SYSTEM Test_7 (* System Configuration *)
  (* Standard: 61499-1 *)
  (* Version 0.3, 2003-12-05, JHC, Rockwell Automation, Renamed from NEWSYSTEM. *)
  (* Version 0.2, 2002-11-05, JHC, Rockwell Automation, Fixed missing (empty) FBD in Application. *)
  (* Version 0.1, 2002-01-17, JHC, Rockwell Automation, Minor cleanup *)
  (* Version 0.0, 2000-05-27, JHC, Rockwell Automation *)
  APPLICATION APP1
  END_APPLICATION
  DEVICE DEV1 : FRAME_DEVICE(BOUNDS := [300,300,300,300], GRID := [1,1])
    RESOURCE RES1 : PANEL_RESOURCE(ROWS := 1, COLS := 1)
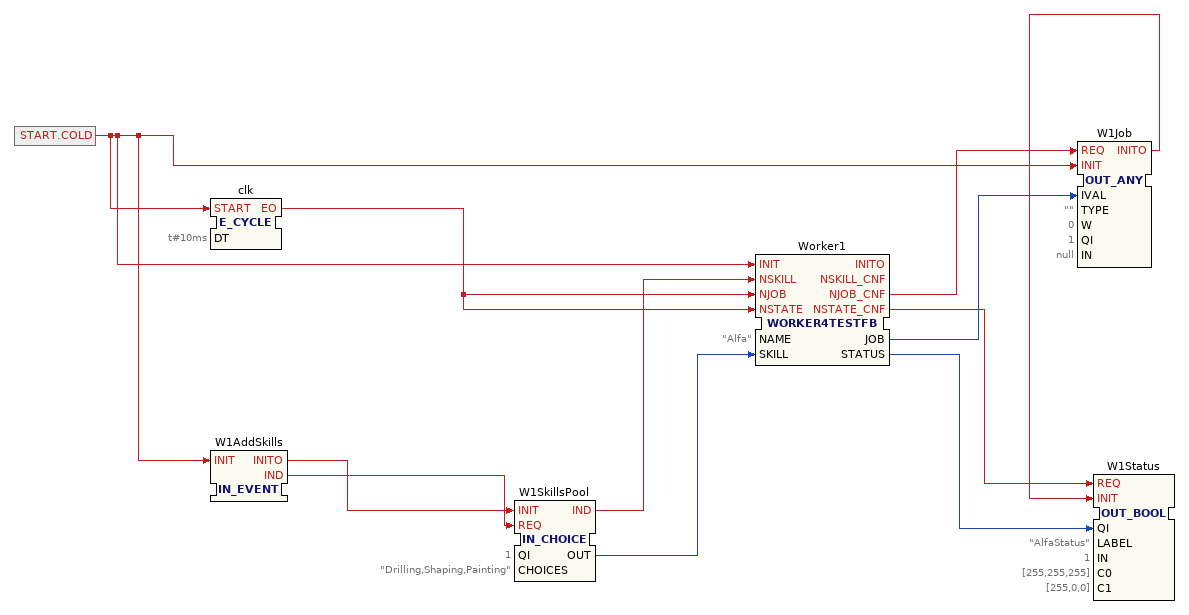
      FBS
        clk : E_CYCLE(DT := t#10ms);
        Worker1 : WORKER4TESTFB(NAME := "Alfa");
        W1Status : OUT_BOOL(LABEL := "AlfaStatus", IN := 1, C0 := [255,255,255], C1 := [255,0,0]);
        W1AddSkills : IN_EVENT;
        W1SkillsPool : IN_CHOICE(QI := 1, CHOICES := "Drilling,Shaping,Painting");
        W1Job : OUT_ANY(TYPE := "", W := 0, QI := 1, IN := null);
      END_FBS
      EVENT_CONNECTIONS
        START.COLD TO clk.START;
        START.COLD TO Worker1.INIT;
        clk.EO TO Worker1.NJOB;
        clk.EO TO Worker1.NSTATE;
        START.COLD TO W1AddSkills.INIT;
        W1AddSkills.INITO TO W1SkillsPool.INIT;
        W1AddSkills.IND TO W1SkillsPool.REQ;
        W1SkillsPool.IND TO Worker1.NSKILL;
        Worker1.NJOB_CNF TO W1Job.REQ;
        START.COLD TO W1Job.INIT;
        Worker1.NSTATE_CNF TO W1Status.REQ;
        W1Job.INITO TO W1Status.INIT;
      END_CONNECTIONS
      DATA_CONNECTIONS
        W1SkillsPool.OUT TO Worker1.SKILL;
        Worker1.JOB TO W1Job.IVAL;
        Worker1.STATUS TO W1Status.QI;
      END_CONNECTIONS
    END_RESOURCE
  END_DEVICE
END_SYSTEM
